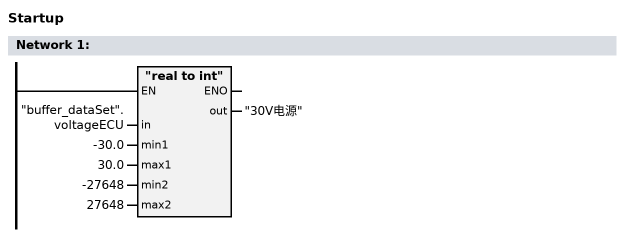
   RUNG wire#powerrail
      "real to int"(in := "buffer_dataSet".voltageECU, min1 := -30.0, max1 := 30.0, min2 := -27648, max2 := 27648, out => "30V电源")
   END_RUNG
   // the same network as SCL:
   "real to int"(in := "buffer_dataSet".voltageECU,
                 min1 := -30.0,
                 max1 := 30.0,
                 min2 := -27648,
                 max2 := 27648,
                 out => "30V电源");
END_REGION
END_ORGANIZATION_BLOCK